FUNCTION_BLOCK FB_Detect_VarChange (* Simple FB with one algorithm *)
  (* Standard: 61499-1 *)
  (* Version 1.0, 2021-08-03, AK121668 *)
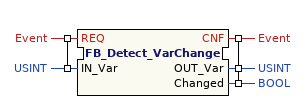
  EVENT_INPUT
    REQ WITH IN_Var; (* Normal Execution Request *)
  END_EVENT
  EVENT_OUTPUT
    CNF WITH OUT_Var, Changed; (* Execution Confirmation *)
  END_EVENT
  VAR_INPUT
    IN_Var : USINT;
  END_VAR
  VAR_OUTPUT
    OUT_Var : USINT;
    Changed : BOOL;
  END_VAR
  VAR
    iValue_Changed : BOOL;
  END_VAR
  ALGORITHM REQ IN ST:
IF OUT_Var <> IN_Var THEN
	iValue_Changed := TRUE;
	OUT_Var := IN_Var;
END_IF;

Changed := iValue_Changed;

IF OUT_Var = IN_Var THEN
	iValue_Changed := FALSE;
END_IF;
  END_ALGORITHM
END_FUNCTION_BLOCK
